(* Logix 5000 project; controller DISPENSE Emulate 5570 rev 36.11; software revision 36.00 *)

TASK MainTask (continuous, watchdog 500 ms) : MainProgram, Model

MODULES
   Local : Emulate 5570 (ICP 2, rev 36.11)
       : 1756-IB16 (ICP 3, rev 3.1, Input RPI 20 ms)
       : vendor 1 type 7 code 16 (ICP 4, rev 3.1, Output RPI 20 ms)
      SENSORS_NET : vendor 1 type 12 code 20 (ICP 5, Ethernet 192.168.0.100, rev 2.1)
         SENSOR : ETHERNET-MODULE (Ethernet 192.168.0.101, rev 1.1, Output RPI 10 ms)
END_MODULES

ADD_ON_INSTRUCTION ANALOG_IN   (* revision 1.0 *)
VAR_INPUT
   Raw_Max : REAL; {required}   // Maximum Bit Value
   Raw_Min : REAL; {required}   // Minimum Bit Value
   EU_Max : REAL; {required}   // Engineering Unit Maximum
   EU_Min : REAL; {required}   // Analog Channel, Source
   Sensor : REAL; {required}   // Analog Channel, Source
END_VAR
VAR_OUTPUT
   EU_Value : REAL; {access Read Only, required}   // Scaled Engineering Unit Value
END_VAR
VAR
   Analog : SCALE; {access None}   // Data Type for Add on Instruction
END_VAR

ROUTINE Logic   (* structured text *)
   Analog.In := Sensor;
   Analog.InRawMax := Raw_Max;
   Analog.InRawMin := Raw_Min;
   Analog.InEUMax := EU_Max;
   Analog.InEUMin := EU_Min;
   SCL(Analog);
   EU_Value := Analog.Out;
END_ROUTINE
END_ADD_ON_INSTRUCTION

VAR_GLOBAL   (* controller tags *)
   DISCHARGE_AUGUR : ALIAS FOR Local:4:O.Data.1;   // Solid Material Discahrge Auger
   DISCHARGE_VALVE : ALIAS FOR Local:4:O.Data.4;   // Discharge Mixture Valve
   DISPENSE_GATE : ALIAS FOR Local:4:O.Data.0;   // Solid Material Dispense Gate
   FLOW_METER : ALIAS FOR SENSOR:I.Data[1];   // Analog Bit Value from Flow Sensor
   FLUID : ANALOG_IN;   // Add on Instruction for Fluid
   FLUID_VALVE : ALIAS FOR Local:4:O.Data.2;   // Dispense Liquid Valve
   FLUID_VOL : DINT;   // Scaled in EU Fluid Valve
   LOAD_CELL : ALIAS FOR SENSOR:I.Data[0];   // Analog Bit Value from weight sensor
   LOW_LEVEL_SW : ALIAS FOR Local:3:I.Data.1;   // Low Level Float Switch, Normally Closed
   MIXER_MOTOR : ALIAS FOR Local:4:O.Data.3;   // Mixer Motor
   SOLID : ANALOG_IN;   // Add on Instruction for Solid
   SOLID_WEIGHT : DINT;   // Scaled in EU Solid Value
   START_PB : ALIAS FOR Local:3:I.Data.0;   // Start Momentary Normally Open Pushbutton
END_VAR

PROGRAM MainProgram   (* main routine MainRoutine *)
VAR
   FLOWMETER_MAX : DINT := 100;   // Maximimum Fluid Setting
   FLOWMETER_MIN : DINT;   // MInimum Fluid Setting
   FLUID_FILLED : BOOL;   // Dispensed from Liquid Valve
   LOAD_CELL_MAX : DINT := 100;   // Maximum Solid Setting
   LOAD_CELL_MIN : DINT;   // Minimum Solid Setting
   MIX_DWELL : TIMER := (PRE := 10000);   // Mixer Motor Timer
   RAW_MAX : DINT := 32767;   // Maximum Bit Value of Sensors
   RAW_MIN : DINT;   // Minimum Bit Value of Sensors
   SOLID_EMPTY : BOOL;   // At Weighting Platform
   SOLID_FILLED : BOOL;   // At Weighting Platform
END_VAR

ROUTINE MainRoutine   (* ladder *)
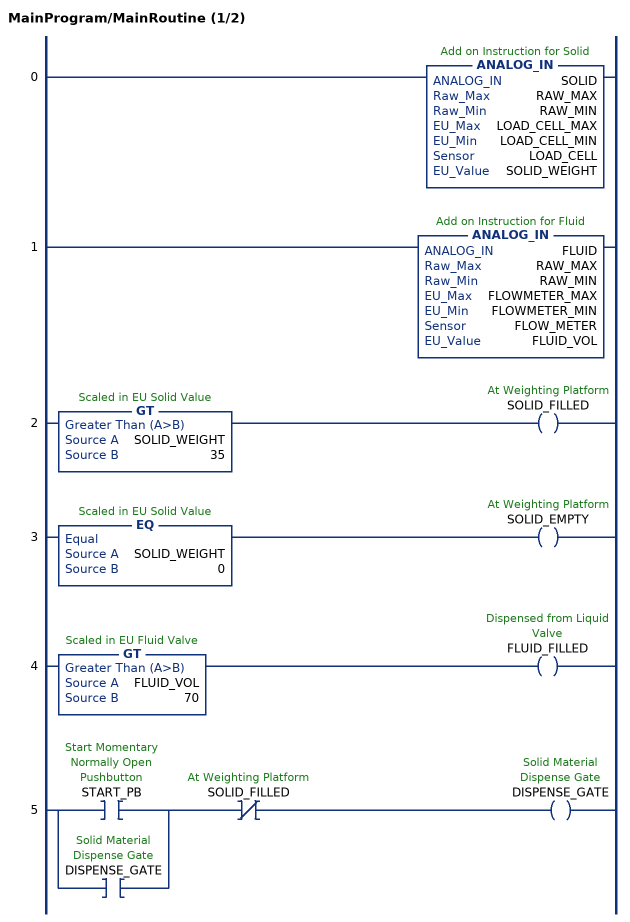
   0: ANALOG_IN(SOLID,RAW_MAX,RAW_MIN,LOAD_CELL_MAX,LOAD_CELL_MIN,LOAD_CELL,SOLID_WEIGHT);
   1: ANALOG_IN(FLUID,RAW_MAX,RAW_MIN,FLOWMETER_MAX,FLOWMETER_MIN,FLOW_METER,FLUID_VOL);
   2: GT(SOLID_WEIGHT,35)OTE(SOLID_FILLED);
   3: EQ(SOLID_WEIGHT,0)OTE(SOLID_EMPTY);
   4: GT(FLUID_VOL,70)OTE(FLUID_FILLED);
   5: [XIC(START_PB) ,XIC(DISPENSE_GATE) ]XIO(SOLID_FILLED)OTE(DISPENSE_GATE);
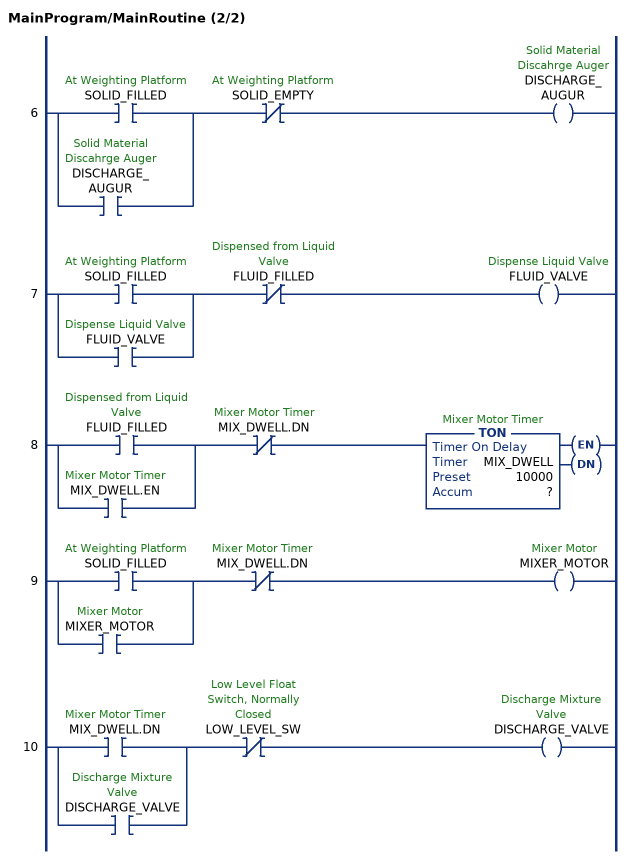
   6: [XIC(SOLID_FILLED) ,XIC(DISCHARGE_AUGUR) ]XIO(SOLID_EMPTY)OTE(DISCHARGE_AUGUR);
   7: [XIC(SOLID_FILLED) ,XIC(FLUID_VALVE) ]XIO(FLUID_FILLED)OTE(FLUID_VALVE);
   8: [XIC(FLUID_FILLED) ,XIC(MIX_DWELL.EN) ]XIO(MIX_DWELL.DN)TON(MIX_DWELL,?,?);
   9: [XIC(SOLID_FILLED) ,XIC(MIXER_MOTOR) ]XIO(MIX_DWELL.DN)OTE(MIXER_MOTOR);
   10: [XIC(MIX_DWELL.DN) ,XIC(DISCHARGE_VALVE) ]XIO(LOW_LEVEL_SW)OTE(DISCHARGE_VALVE);
END_ROUTINE
END_PROGRAM

PROGRAM Model   (* main routine Emulation *)
VAR
   AUGUR_DWELL : TIMER := (PRE := 20);
   DISCHARGE_DWELL : TIMER := (PRE := 5000);
   DISPENSE_DWELL : TIMER := (PRE := 30);
   FLUID_DWELL : TIMER := (PRE := 20);
   LOW_LEVEL_DWELL : TIMER := (PRE := 1000);
END_VAR

ROUTINE Emulation   (* ladder *)
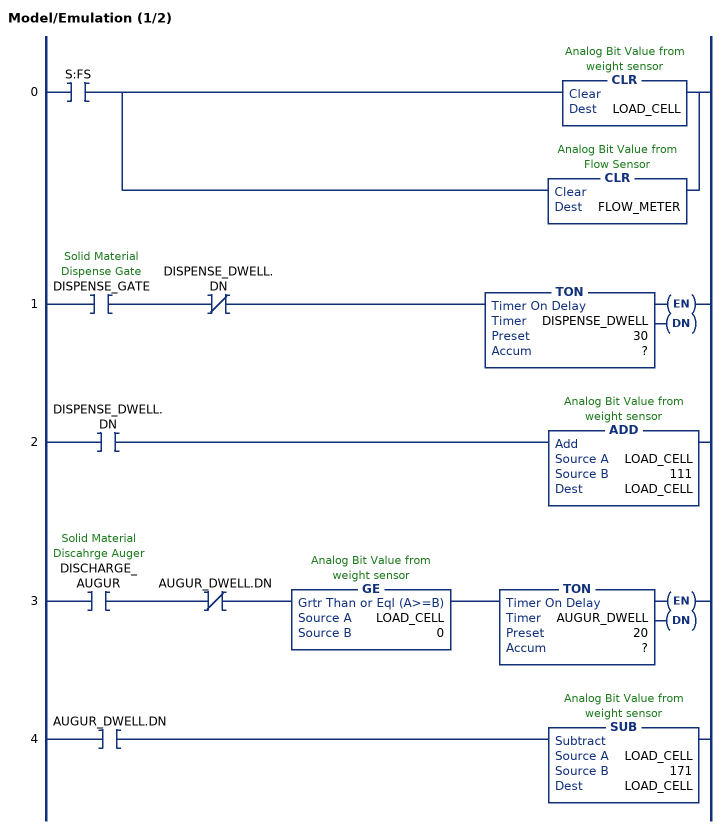
   0: XIC(S:FS)[CLR(LOAD_CELL) ,CLR(FLOW_METER) ];
   1: XIC(DISPENSE_GATE)XIO(DISPENSE_DWELL.DN)TON(DISPENSE_DWELL,?,?);
   2: XIC(DISPENSE_DWELL.DN)ADD(LOAD_CELL,111,LOAD_CELL);
   3: XIC(DISCHARGE_AUGUR)XIO(AUGUR_DWELL.DN)GE(LOAD_CELL,0)TON(AUGUR_DWELL,?,?);
   4: XIC(AUGUR_DWELL.DN)SUB(LOAD_CELL,171,LOAD_CELL);
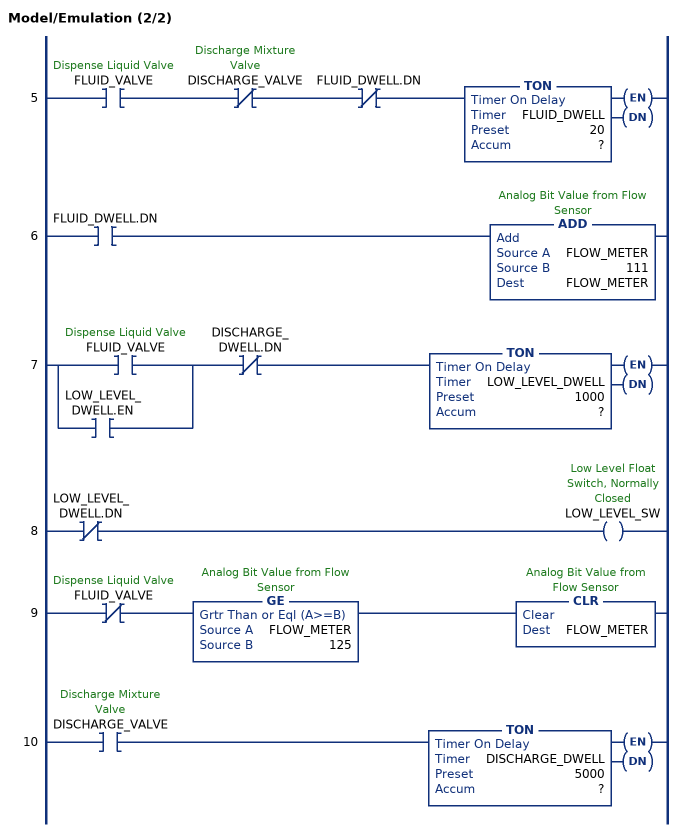
   5: XIC(FLUID_VALVE)XIO(DISCHARGE_VALVE)XIO(FLUID_DWELL.DN)TON(FLUID_DWELL,?,?);
   6: XIC(FLUID_DWELL.DN)ADD(FLOW_METER,111,FLOW_METER);
   7: [XIC(FLUID_VALVE) ,XIC(LOW_LEVEL_DWELL.EN) ]XIO(DISCHARGE_DWELL.DN)TON(LOW_LEVEL_DWELL,?,?);
   8: XIO(LOW_LEVEL_DWELL.DN)OTE(LOW_LEVEL_SW);
   9: XIO(FLUID_VALVE)GE(FLOW_METER,125)CLR(FLOW_METER);
   10: XIC(DISCHARGE_VALVE)TON(DISCHARGE_DWELL,?,?);
END_ROUTINE
END_PROGRAM
